// TIA Portal project "FactoryIO_Template_S7-1200_V16_V16" (V16)
// Vorlageprojekt für das Buch mit Zielsystem S7-1200

(* hardware
DEVICE "S7-1200-Station_1"  S7-1200 Station
   slot 0: "Baugruppenträger_0"  Rack  V1.0
   slot 1: "PLC_1"  CPU 1212C DC/DC/DC  6ES7 212-1AE40-0XB0  V4.4
*)

// ===== PLC "PLC_1"  CPU 1212C DC/DC/DC =====

VAR_GLOBAL   // PLC tag table "Standard-Variablentabelle"
   "START" AT %I0.0 : Bool;
   "RESET" AT %I0.1 : Bool;
   "STOP" AT %I0.2 : Bool;
   "RUNNING" AT %I0.3 : Bool;
   "LEVEL" AT %ID30 : Real;
   "FLOW" AT %ID34 : Real;
   "SETPOINT" AT %ID38 : Real;
   "START LIGHT" AT %Q0.0 : Bool;
   "RESET LIGHT" AT %Q0.1 : Bool;
   "STOP LIGHT" AT %Q0.2 : Bool;
   "FILL VALVE" AT %QD30 : Real;
   "DIS_VALVE" AT %QD34 : Real;
   "SP" AT %QD38 : DInt;
   "PV" AT %QD42 : DInt;
   "FV" AT %QD46 : DInt;
   "SP_PID" AT %ID300 : Real;
   "PV_PID" AT %ID304 : Real;
   "Tag_1" AT %MD300 : Real;
   "Tag_2" AT %QW30 : Word;
END_VAR

DATA_BLOCK "SP_DB"   // DB2
{ S7_Optimized_Access := 'TRUE' }
VERSION : 0.1
// stored: InstanceOfName SENSOR
"SENSOR"
BEGIN
END_DATA_BLOCK

DATA_BLOCK "LEVEL_DB"   // DB3
{ S7_Optimized_Access := 'TRUE' }
VERSION : 0.1
// stored: InstanceOfName SENSOR
"SENSOR"
BEGIN
END_DATA_BLOCK

DATA_BLOCK "FLOW_DB"   // DB4
{ S7_Optimized_Access := 'TRUE' }
VERSION : 0.1
// stored: InstanceOfName SENSOR
"SENSOR"
BEGIN
END_DATA_BLOCK

FUNCTION_BLOCK "SENSOR"   // FB1, LAD
{ S7_Optimized_Access := 'TRUE' }
VERSION : 0.1
   VAR_INPUT
      INPUT : Real;
   END_VAR
   VAR_OUTPUT
      OUTPUT : Real;
   END_VAR
   VAR
      STATIC : Real;
      STATIC_1 : Real;
      STATIC_2 : Real;
      STATIC_3 : Real;
   END_VAR
BEGIN

REGION Network 1
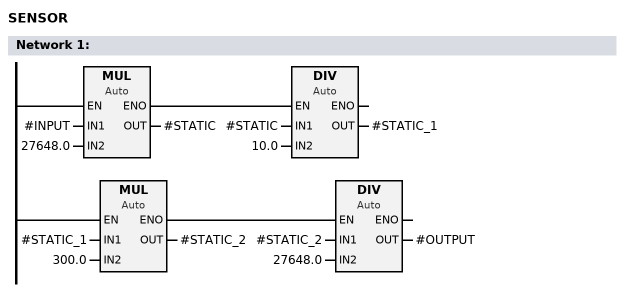
   RUNG wire#powerrail
      Mul(in1 := #INPUT, in2 := 27648.0, out => #STATIC)
      Div(in1 := #STATIC, in2 := 10.0, out => #STATIC_1)
   END_RUNG
   RUNG wire#powerrail
      Mul(in1 := #STATIC_1, in2 := 300.0, out => #STATIC_2)
      Div(in1 := #STATIC_2, in2 := 27648.0, out => #OUTPUT)
   END_RUNG
   // the same network as SCL:
   #STATIC := #INPUT * 27648.0;
   #STATIC_1 := #STATIC / 10.0;
   #STATIC_2 := #STATIC_1 * 300.0;
   #OUTPUT := #STATIC_2 / 27648.0;
END_REGION
END_FUNCTION_BLOCK

FUNCTION "FILL_VLAVE" : Void   // FC1, LAD
{ S7_Optimized_Access := 'TRUE' }
VERSION : 0.1
   VAR_INPUT
      INPUT : Real;
   END_VAR
   VAR_OUTPUT
      OUTPUT : Real;
   END_VAR
   VAR_IN_OUT
      InOut_1 : Real;
   END_VAR
BEGIN

REGION Network 1
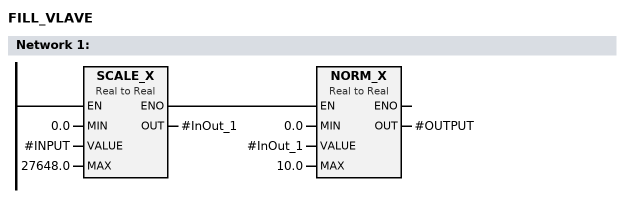
   RUNG wire#powerrail
      { S7_Templates := "[SrcType := Real, DestType := Real]" } Scale(min := 0.0, value := #INPUT, max := 27648.0, out => #InOut_1)
      { S7_Templates := "[SrcType := Real, DestType := Real]" } Normalize(min := 0.0, value := #InOut_1, max := 10.0, out => #OUTPUT)
   END_RUNG
   // the same network as SCL:
   #InOut_1 := SCALE_X(MIN := 0.0, VALUE := #INPUT, MAX := 27648.0);
   #OUTPUT := NORM_X(MIN := 0.0, VALUE := #InOut_1, MAX := 10.0);
END_REGION
END_FUNCTION

FUNCTION "MHJ-PLC-Lab-Function-S71200" : Void   // FC9000, SCL
{ S7_Optimized_Access := 'TRUE' }
VERSION : 0.1
   VAR_TEMP
      rdTimeReturn : Int;
      outputTime : DTL;
      SyncVal : Byte;
      forVal : Int;
      forVal_2 : Int;
      Value : Byte;
   END_VAR
   VAR CONSTANT
      CompVal : Byte := 16#34;
      Value_01 : Byte := 16#11;
      Value_01_DW : DWord := 16#A165_D992;
      Value_02_DW : DWord := 16#58BE_4401;
   END_VAR
BEGIN

   #Value:=PEEK(area := 16#82,
        dbNumber := 0,
        byteOffset := 511);
   #Value := #Value + 1;

   POKE(area := 16#82,
        dbNumber := 0,
        byteOffset := 511,
        value := #Value);

   POKE(area:=16#81,
        dbNumber:=0,
        byteOffset:=1016,
        value:=#Value_01_DW);
   POKE(area := 16#81,
        dbNumber := 0,
        byteOffset := 1020,
        value := #Value_02_DW);

   POKE(area := 16#81,
        dbNumber := 0,
        byteOffset := 511,
        value := B#16#00);

   FOR #forVal := 0 TO 120 DO
       FOR #forVal_2:=0 TO 10 DO
           #rdTimeReturn:=RD_SYS_T(#outputTime);
           #rdTimeReturn := WR_SYS_T(#outputTime);
           #rdTimeReturn := RD_SYS_T(#outputTime);
           #rdTimeReturn := WR_SYS_T(#outputTime);
       END_FOR;
       #SyncVal:= PEEK(area := 16#81,
                      dbNumber := 0,
                      byteOffset := 511);
       IF #SyncVal = #CompVal THEN
          GOTO M_1;
       END_IF;
   END_FOR;
   RETURN;

   M_1:
   POKE(area := 16#81,
        dbNumber := 0,
        byteOffset := 511,
        value := B#16#0);
END_FUNCTION

ORGANIZATION_BLOCK "Main"   // OB1, LAD, ProgramCycle
TITLE = "Main Program Sweep (Cycle)"
{ S7_Optimized_Access := 'TRUE' }
VERSION : 0.1
   VAR_INPUT
      Initial_Call : Bool;   // Initial call of this OB
      Remanence : Bool;   // =True, if remanent data are available
   END_VAR
   VAR_TEMP   // added for the SCL form of the ladder/FBD networks
      _w1 : Bool;
   END_VAR
BEGIN

REGION Network 1: Konnektierungsbaustein für PLC-Lab
   // Im Netzwerk 1 wird der Konnektierungsbaustein für PLC-Lab aufgerufen.
   // Dieser Aufruf darf nicht entfernt werden!
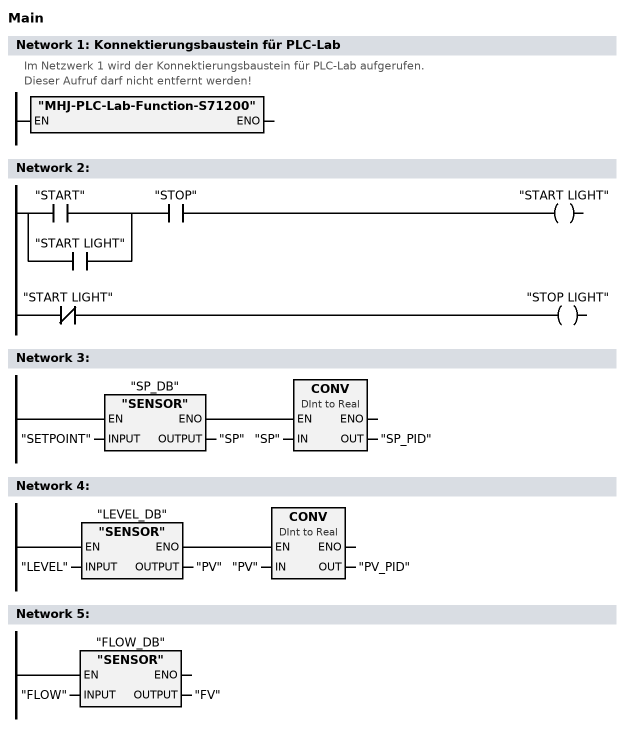
   RUNG wire#powerrail
      "MHJ-PLC-Lab-Function-S71200"()
   END_RUNG
   // the same network as SCL:
   "MHJ-PLC-Lab-Function-S71200"();
END_REGION

REGION Network 2
   RUNG wire#powerrail
      Contact( "START" )
      wire#w1
      Contact( "STOP" )
      Coil( "START LIGHT" )
   END_RUNG
   RUNG wire#powerrail
      Contact( "START LIGHT" )
   END_RUNG wire#w1
   RUNG wire#powerrail
      I_Contact( "START LIGHT" )
      Coil( "STOP LIGHT" )
   END_RUNG
   // the same network as SCL:
   "START LIGHT" := ("START" OR "START LIGHT") AND "STOP";
   "STOP LIGHT" := NOT "START LIGHT";
END_REGION

REGION Network 3
   RUNG wire#powerrail
      "SP_DB"(INPUT := "SETPOINT", OUTPUT => "SP")
      { S7_Templates := "[SrcType := DInt, DestType := Real]" } Convert(in := "SP", out => "SP_PID")
   END_RUNG
   // the same network as SCL:
   "SP_DB"(INPUT := "SETPOINT", OUTPUT => "SP", ENO => #_w1);   // "SENSOR"
   IF #_w1 THEN "SP_PID" := DINT_TO_REAL("SP"); END_IF;
END_REGION

REGION Network 4
   RUNG wire#powerrail
      "LEVEL_DB"(INPUT := "LEVEL", OUTPUT => "PV")
      { S7_Templates := "[SrcType := DInt, DestType := Real]" } Convert(in := "PV", out => "PV_PID")
   END_RUNG
   // the same network as SCL:
   "LEVEL_DB"(INPUT := "LEVEL", OUTPUT => "PV", ENO => #_w1);   // "SENSOR"
   IF #_w1 THEN "PV_PID" := DINT_TO_REAL("PV"); END_IF;
END_REGION

REGION Network 5
   RUNG wire#powerrail
      "FLOW_DB"(INPUT := "FLOW", OUTPUT => "FV")
   END_RUNG
   // the same network as SCL:
   "FLOW_DB"(INPUT := "FLOW", OUTPUT => "FV");   // "SENSOR"
END_REGION
END_ORGANIZATION_BLOCK

ORGANIZATION_BLOCK "Cyclic interrupt"   // OB30, LAD, CyclicInterrupt
{ S7_Optimized_Access := 'TRUE' }
VERSION : 0.1
   VAR_INPUT
      Initial_Call : Bool;   // Initial call of this OB
      Event_Count : Int;   // Events discarded
   END_VAR
BEGIN

REGION Network 1
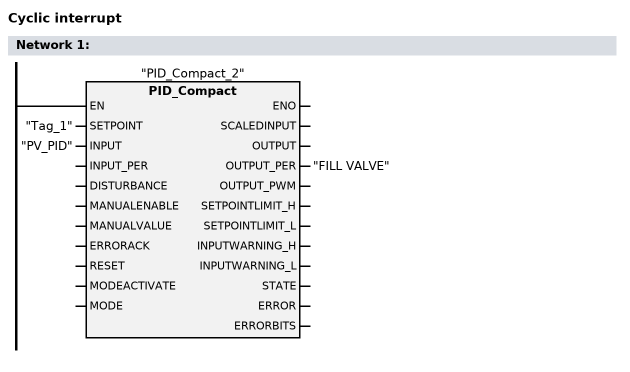
   "PID_Compact_2"(Setpoint := "Tag_1", Input := "PV_PID", Output_PER => "FILL VALVE");   // PID_Compact
END_REGION
END_ORGANIZATION_BLOCK